(* IEC 61131-3 sources: s22-soft-shell/st_interpret/tests/test_inputs/execution/st_subset_7, 8 files *)

(* ---- 07_Equality.st ---- *)
PROGRAM 07_Equality
    VAR
		a : bool;
		b : bool;
		c : bool;
		d : bool;
        ST_TESTING_RESULT : bool;
    END_VAR
		a := TRUE = False; // Result = False
		b := false <> true; // Result = True
		c := False = FALSE; // Result = True
		d := tRuE <> True; // Result = False
        ST_TESTING_RESULT := (not a & b) & (c & not d);
END_PROGRAM

(* ---- 07_Greater_Eq.st ---- *)
PROGRAM 07_Greater_Eq
    VAR
		a : bool;
		b : bool;
		c : bool;
		d : bool;
        ST_TESTING_RESULT : bool;
    END_VAR
		a := 8 >= -5; // Result = True
		b := -4 >= -4; // Result = True
		c := 0 >= 5555; // Result = False
		d := -34 >= -55; // Result = True
        ST_TESTING_RESULT := (a & b) & (not c & d);
END_PROGRAM

(* ---- 07_Greater_Than.st ---- *)
PROGRAM 07_Greater_Than
    VAR
		a : bool;
		b : bool;
		c : bool;
		d : bool;
        ST_TESTING_RESULT : bool;
    END_VAR
		a := 8 > -5; // Result = True
		b := -4 > -4; // Result = False
		c := 0 > 5555; // Result = False
		d := -34 > -55; // Result = True
        ST_TESTING_RESULT := (a & not b) & (not c & d);
END_PROGRAM

(* ---- 07_Less_Eq.st ---- *)
PROGRAM 07_Less_Eq
    VAR
		a : bool;
		b : bool;
		c : bool;
		d : bool;
        ST_TESTING_RESULT : bool;
    END_VAR
		a := 8 <= -5; // Result = False
		b := 44 <= 44; // Result = True
		c := 0 <= 5555; // Result = True
		d := -34 <= -55; // Result = False
        ST_TESTING_RESULT := (not a & b) & (c & not d);
END_PROGRAM

(* ---- 07_Less_Than.st ---- *)
PROGRAM 07_Less_Eq
    VAR
		a : bool;
		b : bool;
		c : bool;
		d : bool;
        ST_TESTING_RESULT : bool;
    END_VAR
		a := 8 < -5; // Result = False
		b := 44 < 44; // Result = False
		c := 0 < 5555; // Result = True
		d := -34 < -55; // Result = False
        ST_TESTING_RESULT := (not a & not b) & (c & not d);
END_PROGRAM

(* ---- 07_Test_A.st ---- *)
PROGRAM 07_Test_A
    VAR
		a : Int;
		b : Int;
		c : bool;
		d : bool;
        ST_TESTING_RESULT : bool;
    END_VAR
		a := 3;
		b := 6;
		c := 3 >= a = 6-20 < 26; // Result = True
		d := (16/4) = (b-4) * 2; // Result = True
        ST_TESTING_RESULT := (a = 3 & b = 6) & (c & d);
END_PROGRAM

(* ---- 07_While.st ---- *)
PROGRAM 07_While
    VAR
		a : Int;
		b : Int;
		ST_TESTING_RESULT : bool;
    END_VAR
		a := 1;
        b := 1;

        WHILE (a < 8) DO
            a := a + 1;

            WHILE (b < 3) DO
                b:= b+1;
            END_WHILE;
        END_WHILE;

        ST_TESTING_RESULT := (a = 8) & (b = 3);
END_PROGRAM

(* ---- 07_While_If.st ---- *)
// Tests that while and IF statements work inside eachother
PROGRAM 07_While_If
    VAR
	a : Int;
        b : Int;
        c : Int;
        d : Int;
        ST_TESTING_RESULT : bool;
    END_VAR
	a := 0;
        b := 0;
        c := 0;
        d := 0;
        WHILE (a < 5) DO
            a := a + 1;
            IF a > 3 THEN
                b := 3;
            END_IF;
        END_WHILE;

        IF (c < 5) THEN
            WHILE (d < 4) DO
                d := d + 1;
            END_WHILE;
            c := 2;
        END_IF;
        ST_TESTING_RESULT := (a = 5 & b = 3) & (c = 2 & d = 4);
END_PROGRAM
